# EPICS autosave request: iocBoot/ioc13PHD2000/auto_settings.req
file "PHD2000_settings.req",         P=$(P), R=$(R)
